// TIA Portal project "automated-warehouse" (V18)
// Vorlageprojekt für das Buch mit Zielsystem S7-1200

(* hardware
DEVICE "S7-1200-Station_1"  S7-1200 Station
   slot 0: "Baugruppenträger_0"  Rack  V1.0
   slot 1: "PLC_1"  CPU 1211C DC/DC/DC  6ES7 211-1AE40-0XB0  V4.1
*)

// ===== PLC "PLC_1"  CPU 1211C DC/DC/DC =====

VAR_GLOBAL   // PLC tag table "Standard-Variablentabelle"
   "Stored Shelf Value" AT %MW0 : Int;
   "Load Sequence Active" AT %M0.1 : Bool;
   "Unload Sequence Active" AT %M0.2 : Bool;
END_VAR

VAR_GLOBAL   // PLC tag table "FactoryIO"
   "Lift" AT %Q0.4 : Bool;
   "Forks Left" AT %Q0.2 : Bool;
   "Forks Right" AT %Q0.3 : Bool;
   "Entry Conveyor" AT %Q0.0 : Bool;
   "Load Conveyor" AT %Q0.1 : Bool;
   "Unload Conveyor" AT %Q0.5 : Bool;
   "Exit Conveyor" AT %Q0.6 : Bool;
   "Start light" AT %Q0.7 : Bool;
   "Stop light" AT %Q1.1 : Bool;
   "Target Position" AT %QD30 : DInt;
   "Reset Light" AT %Q1.0 : Bool;
   "At Entry" AT %I0.0 : Bool;
   "At Load" AT %I0.1 : Bool;
   "At Left" AT %I0.2 : Bool;
   "At Middle" AT %I0.3 : Bool;
   "At Right" AT %I0.4 : Bool;
   "At Unload" AT %I0.5 : Bool;
   "At Exit" AT %I0.6 : Bool;
   "Moving X" AT %I0.7 : Bool;
   "Moving Z" AT %I1.0 : Bool;
   "Start" AT %I1.1 : Bool;
   "Reset" AT %I1.2 : Bool;
   "Stop" AT %I1.3 : Bool;
   "Emergency stop" AT %I1.4 : Bool;
   "Load mode" AT %I1.5 : Bool;
END_VAR

DATA_BLOCK "Stacker Crane_DB"   // DB1
{ S7_Optimized_Access := 'TRUE' }
VERSION : 0.1
// stored: InstanceOfName Stacker Crane
"Stacker Crane"
BEGIN
END_DATA_BLOCK

DATA_BLOCK "Control Panel_DB"   // DB2
{ S7_Optimized_Access := 'TRUE' }
VERSION : 0.1
// stored: InstanceOfName Control Panel
"Control Panel"
BEGIN
END_DATA_BLOCK

DATA_BLOCK "Conveyors_DB"   // DB3
{ S7_Optimized_Access := 'TRUE' }
VERSION : 0.1
// stored: InstanceOfName Conveyors
"Conveyors"
BEGIN
END_DATA_BLOCK

// folder: System blocks/Program resources

DATA_BLOCK "IEC_Timer_0_DB"   // DB4
{ S7_Optimized_Access := 'TRUE' }
AUTHOR : Simatic
FAMILY : IEC
NAME : IEC_TMR
VERSION : 1.0
// stored: InstanceOfName IEC_TIMER
"IEC_TIMER"
BEGIN
END_DATA_BLOCK

DATA_BLOCK "IEC_Timer_0_DB_1"   // DB5
{ S7_Optimized_Access := 'TRUE' }
AUTHOR : Simatic
FAMILY : IEC
NAME : IEC_TMR
VERSION : 1.0
// stored: InstanceOfName IEC_TIMER
"IEC_TIMER"
BEGIN
END_DATA_BLOCK

// folder: (top level)

FUNCTION_BLOCK "Stacker Crane"   // FB1, LAD
{ S7_Optimized_Access := 'TRUE' }
VERSION : 0.1
   VAR_INPUT
      "Moving X" : Bool;
      "Moving Z" : Bool;
      "At Entry" : Bool;
      "At Load" : Bool;
      "At Unload" : Bool;
      "At Left" : Bool;
      "At Middle" : Bool;
      "At Right" : Bool;
      "Load mode" : Bool;
      Reset : Bool;
      "Start light" : Bool;
      "Emergency Stop" : Bool;
   END_VAR
   VAR_OUTPUT
      Lift : Bool;
      "Forks Left" : Bool;
      "Forks Right" : Bool;
      "Target Position" : DInt;
      "Stored Shelf Value" : Int;
      "Load Sequence Active" : Bool;
      "Unload Sequence Active" : Bool;
   END_VAR
   VAR
      n_trig : Array[0..10] of Bool;
      "Step" : Int := 0;
   END_VAR
   VAR_TEMP   // added for the SCL form of the ladder/FBD networks
      _w1 : Bool;
      _w2 : Bool;
      _w3 : Bool;
   END_VAR
BEGIN

REGION Network 1: <-------------------------- Load Section -------------------------->
END_REGION

REGION Network 2: Step 0 - Start Load Sequence
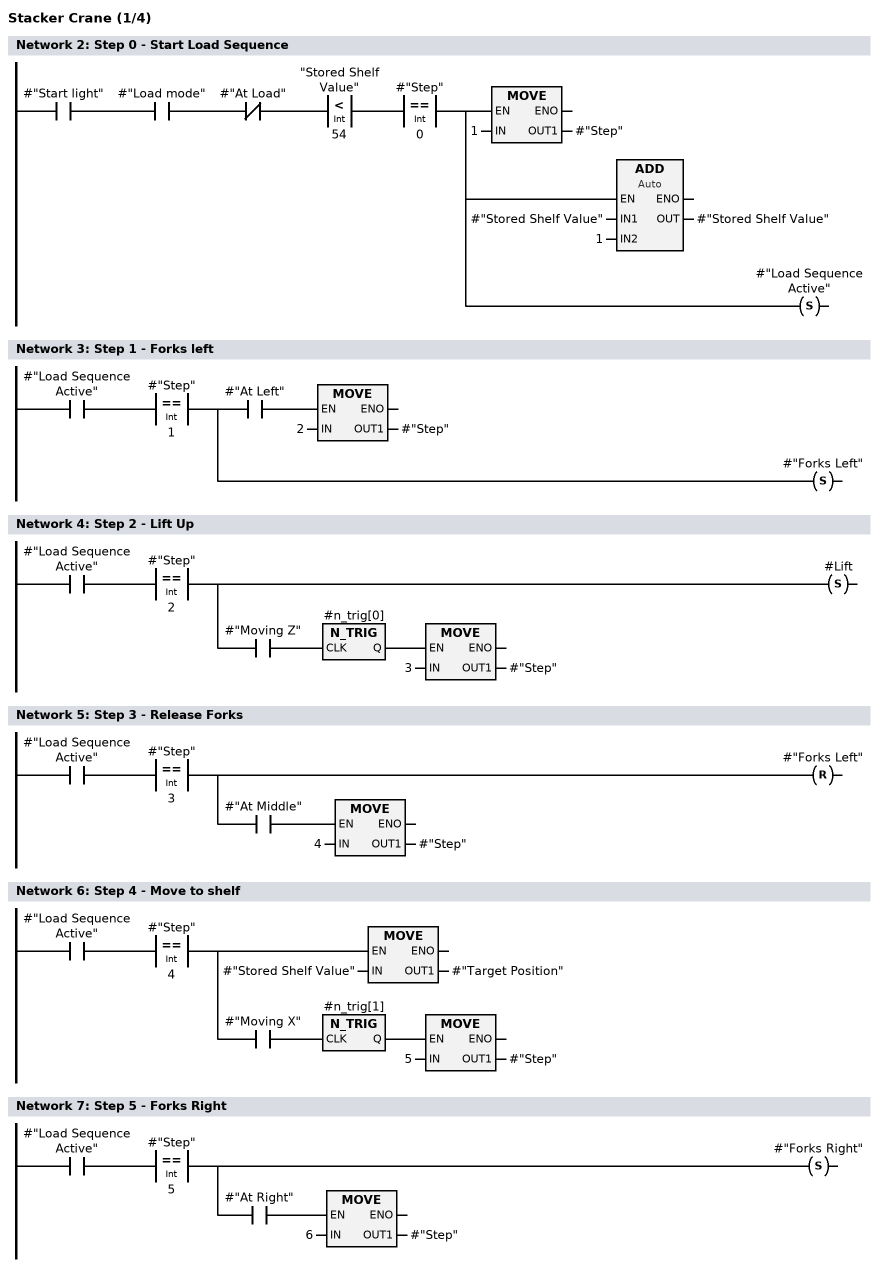
   RUNG wire#powerrail
      Contact( #"Start light" )
      Contact( #"Load mode" )
      I_Contact( #"At Load" )
      { S7_Templates := "SrcType := Int" } LT_Contact(in1 := "Stored Shelf Value", in2 := 54)
      { S7_Templates := "SrcType := Int" } EQ_Contact(in1 := #"Step", in2 := 0)
      wire#w1
      Move(in := 1, out1 => #"Step")
   END_RUNG
   RUNG wire#w1
      Add(in1 := #"Stored Shelf Value", in2 := 1, out => #"Stored Shelf Value")
   END_RUNG
   RUNG wire#w1
      S_Coil( #"Load Sequence Active" )
   END_RUNG
   // the same network as SCL:
   #_w1 := #"Start light" AND #"Load mode" AND NOT #"At Load" AND ("Stored Shelf Value" < 54) AND (#"Step" = 0);
   IF #_w1 THEN
       #"Step" := 1;
       #"Stored Shelf Value" := #"Stored Shelf Value" + 1;
       #"Load Sequence Active" := TRUE;
   END_IF;
END_REGION

REGION Network 3: Step 1 - Forks left
   RUNG wire#powerrail
      Contact( #"Load Sequence Active" )
      { S7_Templates := "SrcType := Int" } EQ_Contact(in1 := #"Step", in2 := 1)
      wire#w1
      Contact( #"At Left" )
      Move(in := 2, out1 => #"Step")
   END_RUNG
   RUNG wire#w1
      S_Coil( #"Forks Left" )
   END_RUNG
   // the same network as SCL:
   #_w1 := #"Load Sequence Active" AND (#"Step" = 1);
   IF #_w1 AND #"At Left" THEN #"Step" := 2; END_IF;
   IF #_w1 THEN #"Forks Left" := TRUE; END_IF;
END_REGION

REGION Network 4: Step 2 - Lift Up
   RUNG wire#powerrail
      Contact( #"Load Sequence Active" )
      { S7_Templates := "SrcType := Int" } EQ_Contact(in1 := #"Step", in2 := 2)
      wire#w1
      S_Coil( #Lift )
   END_RUNG
   RUNG wire#w1
      Contact( #"Moving Z" )
      N_Trig( #n_trig[0] )
      Move(in := 3, out1 => #"Step")
   END_RUNG
   // the same network as SCL:
   #_w1 := #"Load Sequence Active" AND (#"Step" = 2);
   IF #_w1 THEN #Lift := TRUE; END_IF;
   #_w2 := #_w1 AND #"Moving Z";
   #_w3 := NOT #_w2 AND #n_trig[0];   // falling edge
   #n_trig[0] := #_w2;
   IF #_w3 THEN #"Step" := 3; END_IF;
END_REGION

REGION Network 5: Step 3 - Release Forks
   RUNG wire#powerrail
      Contact( #"Load Sequence Active" )
      { S7_Templates := "SrcType := Int" } EQ_Contact(in1 := #"Step", in2 := 3)
      wire#w1
      R_Coil( #"Forks Left" )
   END_RUNG
   RUNG wire#w1
      Contact( #"At Middle" )
      Move(in := 4, out1 => #"Step")
   END_RUNG
   // the same network as SCL:
   #_w1 := #"Load Sequence Active" AND (#"Step" = 3);
   IF #_w1 THEN #"Forks Left" := FALSE; END_IF;
   IF #_w1 AND #"At Middle" THEN #"Step" := 4; END_IF;
END_REGION

REGION Network 6: Step 4 - Move to shelf
   RUNG wire#powerrail
      Contact( #"Load Sequence Active" )
      { S7_Templates := "SrcType := Int" } EQ_Contact(in1 := #"Step", in2 := 4)
      wire#w1
      Move(in := #"Stored Shelf Value", out1 => #"Target Position")
   END_RUNG
   RUNG wire#w1
      Contact( #"Moving X" )
      N_Trig( #n_trig[1] )
      Move(in := 5, out1 => #"Step")
   END_RUNG
   // the same network as SCL:
   #_w1 := #"Load Sequence Active" AND (#"Step" = 4);
   IF #_w1 THEN #"Target Position" := #"Stored Shelf Value"; END_IF;
   #_w2 := #_w1 AND #"Moving X";
   #_w3 := NOT #_w2 AND #n_trig[1];   // falling edge
   #n_trig[1] := #_w2;
   IF #_w3 THEN #"Step" := 5; END_IF;
END_REGION

REGION Network 7: Step 5 - Forks Right
   RUNG wire#powerrail
      Contact( #"Load Sequence Active" )
      { S7_Templates := "SrcType := Int" } EQ_Contact(in1 := #"Step", in2 := 5)
      wire#w1
      S_Coil( #"Forks Right" )
   END_RUNG
   RUNG wire#w1
      Contact( #"At Right" )
      Move(in := 6, out1 => #"Step")
   END_RUNG
   // the same network as SCL:
   #_w1 := #"Load Sequence Active" AND (#"Step" = 5);
   IF #_w1 THEN #"Forks Right" := TRUE; END_IF;
   IF #_w1 AND #"At Right" THEN #"Step" := 6; END_IF;
END_REGION

REGION Network 8: Step 6 - Release Lift
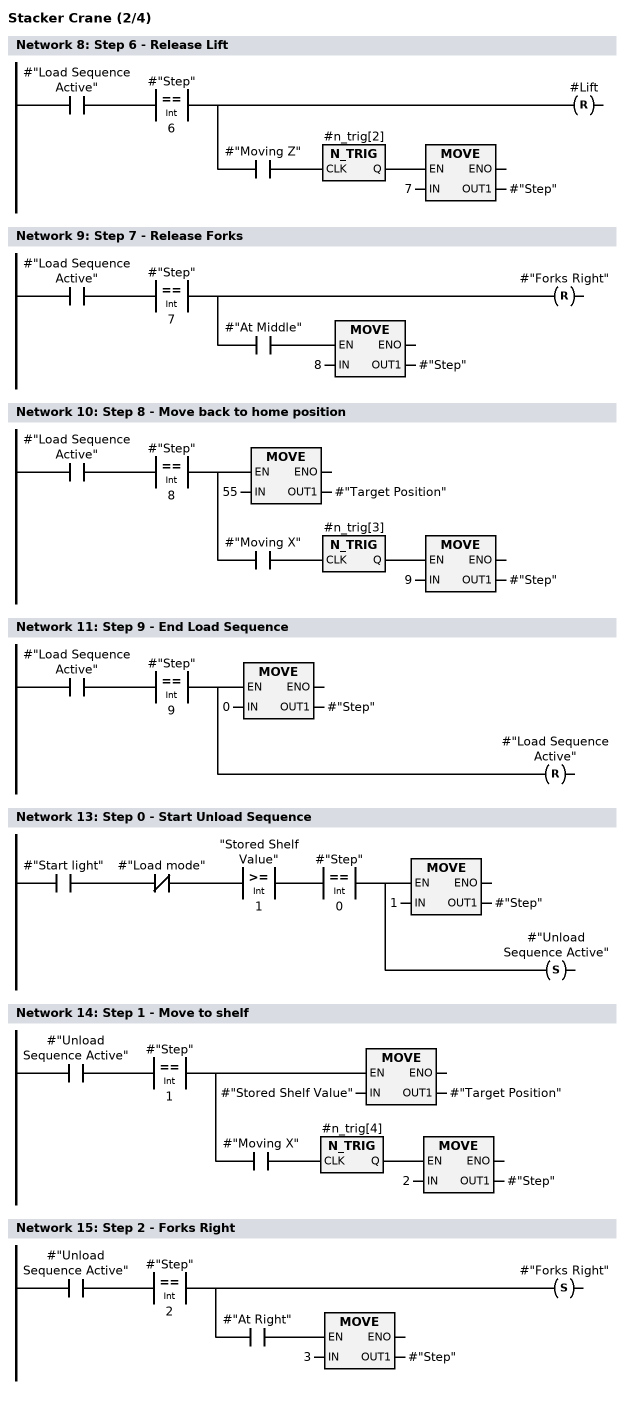
   RUNG wire#powerrail
      Contact( #"Load Sequence Active" )
      { S7_Templates := "SrcType := Int" } EQ_Contact(in1 := #"Step", in2 := 6)
      wire#w1
      R_Coil( #Lift )
   END_RUNG
   RUNG wire#w1
      Contact( #"Moving Z" )
      N_Trig( #n_trig[2] )
      Move(in := 7, out1 => #"Step")
   END_RUNG
   // the same network as SCL:
   #_w1 := #"Load Sequence Active" AND (#"Step" = 6);
   IF #_w1 THEN #Lift := FALSE; END_IF;
   #_w2 := #_w1 AND #"Moving Z";
   #_w3 := NOT #_w2 AND #n_trig[2];   // falling edge
   #n_trig[2] := #_w2;
   IF #_w3 THEN #"Step" := 7; END_IF;
END_REGION

REGION Network 9: Step 7 - Release Forks
   RUNG wire#powerrail
      Contact( #"Load Sequence Active" )
      { S7_Templates := "SrcType := Int" } EQ_Contact(in1 := #"Step", in2 := 7)
      wire#w1
      R_Coil( #"Forks Right" )
   END_RUNG
   RUNG wire#w1
      Contact( #"At Middle" )
      Move(in := 8, out1 => #"Step")
   END_RUNG
   // the same network as SCL:
   #_w1 := #"Load Sequence Active" AND (#"Step" = 7);
   IF #_w1 THEN #"Forks Right" := FALSE; END_IF;
   IF #_w1 AND #"At Middle" THEN #"Step" := 8; END_IF;
END_REGION

REGION Network 10: Step 8 - Move back to home position
   RUNG wire#powerrail
      Contact( #"Load Sequence Active" )
      { S7_Templates := "SrcType := Int" } EQ_Contact(in1 := #"Step", in2 := 8)
      wire#w1
      Move(in := 55, out1 => #"Target Position")
   END_RUNG
   RUNG wire#w1
      Contact( #"Moving X" )
      N_Trig( #n_trig[3] )
      Move(in := 9, out1 => #"Step")
   END_RUNG
   // the same network as SCL:
   #_w1 := #"Load Sequence Active" AND (#"Step" = 8);
   IF #_w1 THEN #"Target Position" := 55; END_IF;
   #_w2 := #_w1 AND #"Moving X";
   #_w3 := NOT #_w2 AND #n_trig[3];   // falling edge
   #n_trig[3] := #_w2;
   IF #_w3 THEN #"Step" := 9; END_IF;
END_REGION

REGION Network 11: Step 9 - End Load Sequence
   RUNG wire#powerrail
      Contact( #"Load Sequence Active" )
      { S7_Templates := "SrcType := Int" } EQ_Contact(in1 := #"Step", in2 := 9)
      wire#w1
      Move(in := 0, out1 => #"Step")
   END_RUNG
   RUNG wire#w1
      R_Coil( #"Load Sequence Active" )
   END_RUNG
   // the same network as SCL:
   #_w1 := #"Load Sequence Active" AND (#"Step" = 9);
   IF #_w1 THEN
       #"Step" := 0;
       #"Load Sequence Active" := FALSE;
   END_IF;
END_REGION

REGION Network 12: <-------------------------- Unload Section -------------------------->
END_REGION

REGION Network 13: Step 0 - Start Unload Sequence
   RUNG wire#powerrail
      Contact( #"Start light" )
      I_Contact( #"Load mode" )
      { S7_Templates := "SrcType := Int" } GE_Contact(in1 := "Stored Shelf Value", in2 := 1)
      { S7_Templates := "SrcType := Int" } EQ_Contact(in1 := #"Step", in2 := 0)
      wire#w1
      Move(in := 1, out1 => #"Step")
   END_RUNG
   RUNG wire#w1
      S_Coil( #"Unload Sequence Active" )
   END_RUNG
   // the same network as SCL:
   #_w1 := #"Start light" AND NOT #"Load mode" AND ("Stored Shelf Value" >= 1) AND (#"Step" = 0);
   IF #_w1 THEN
       #"Step" := 1;
       #"Unload Sequence Active" := TRUE;
   END_IF;
END_REGION

REGION Network 14: Step 1 - Move to shelf
   RUNG wire#powerrail
      Contact( #"Unload Sequence Active" )
      { S7_Templates := "SrcType := Int" } EQ_Contact(in1 := #"Step", in2 := 1)
      wire#w1
      Move(in := #"Stored Shelf Value", out1 => #"Target Position")
   END_RUNG
   RUNG wire#w1
      Contact( #"Moving X" )
      N_Trig( #n_trig[4] )
      Move(in := 2, out1 => #"Step")
   END_RUNG
   // the same network as SCL:
   #_w1 := #"Unload Sequence Active" AND (#"Step" = 1);
   IF #_w1 THEN #"Target Position" := #"Stored Shelf Value"; END_IF;
   #_w2 := #_w1 AND #"Moving X";
   #_w3 := NOT #_w2 AND #n_trig[4];   // falling edge
   #n_trig[4] := #_w2;
   IF #_w3 THEN #"Step" := 2; END_IF;
END_REGION

REGION Network 15: Step 2 - Forks Right
   RUNG wire#powerrail
      Contact( #"Unload Sequence Active" )
      { S7_Templates := "SrcType := Int" } EQ_Contact(in1 := #"Step", in2 := 2)
      wire#w1
      S_Coil( #"Forks Right" )
   END_RUNG
   RUNG wire#w1
      Contact( #"At Right" )
      Move(in := 3, out1 => #"Step")
   END_RUNG
   // the same network as SCL:
   #_w1 := #"Unload Sequence Active" AND (#"Step" = 2);
   IF #_w1 THEN #"Forks Right" := TRUE; END_IF;
   IF #_w1 AND #"At Right" THEN #"Step" := 3; END_IF;
END_REGION

REGION Network 16: Step 3 - Lift Up
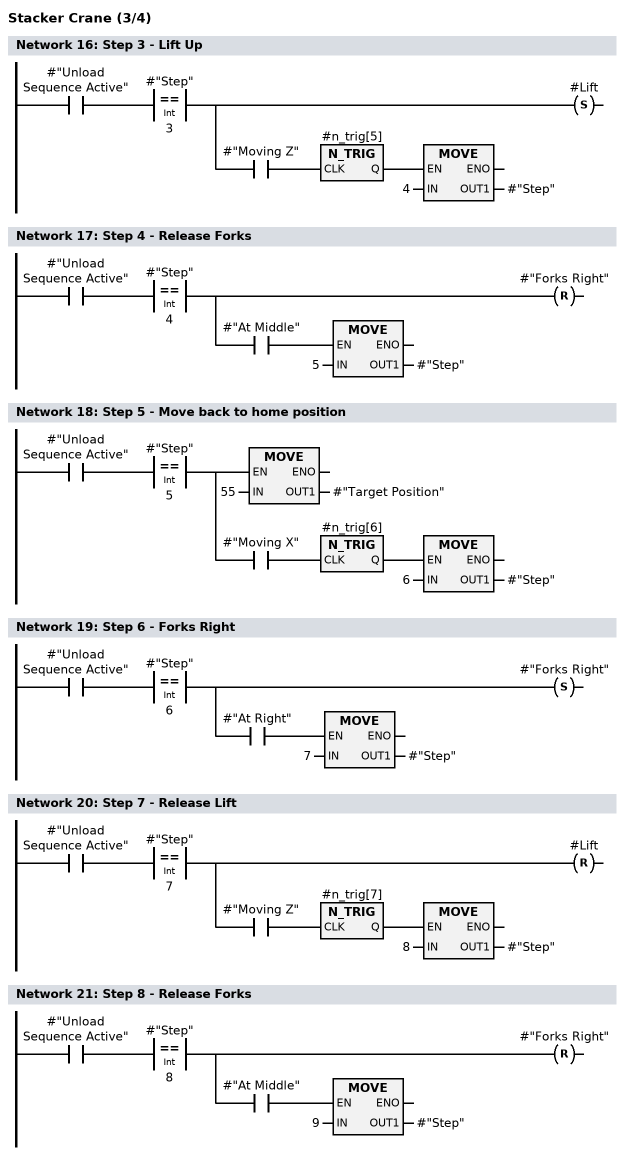
   RUNG wire#powerrail
      Contact( #"Unload Sequence Active" )
      { S7_Templates := "SrcType := Int" } EQ_Contact(in1 := #"Step", in2 := 3)
      wire#w1
      S_Coil( #Lift )
   END_RUNG
   RUNG wire#w1
      Contact( #"Moving Z" )
      N_Trig( #n_trig[5] )
      Move(in := 4, out1 => #"Step")
   END_RUNG
   // the same network as SCL:
   #_w1 := #"Unload Sequence Active" AND (#"Step" = 3);
   IF #_w1 THEN #Lift := TRUE; END_IF;
   #_w2 := #_w1 AND #"Moving Z";
   #_w3 := NOT #_w2 AND #n_trig[5];   // falling edge
   #n_trig[5] := #_w2;
   IF #_w3 THEN #"Step" := 4; END_IF;
END_REGION

REGION Network 17: Step 4 - Release Forks
   RUNG wire#powerrail
      Contact( #"Unload Sequence Active" )
      { S7_Templates := "SrcType := Int" } EQ_Contact(in1 := #"Step", in2 := 4)
      wire#w1
      R_Coil( #"Forks Right" )
   END_RUNG
   RUNG wire#w1
      Contact( #"At Middle" )
      Move(in := 5, out1 => #"Step")
   END_RUNG
   // the same network as SCL:
   #_w1 := #"Unload Sequence Active" AND (#"Step" = 4);
   IF #_w1 THEN #"Forks Right" := FALSE; END_IF;
   IF #_w1 AND #"At Middle" THEN #"Step" := 5; END_IF;
END_REGION

REGION Network 18: Step 5 - Move back to home position
   RUNG wire#powerrail
      Contact( #"Unload Sequence Active" )
      { S7_Templates := "SrcType := Int" } EQ_Contact(in1 := #"Step", in2 := 5)
      wire#w1
      Move(in := 55, out1 => #"Target Position")
   END_RUNG
   RUNG wire#w1
      Contact( #"Moving X" )
      N_Trig( #n_trig[6] )
      Move(in := 6, out1 => #"Step")
   END_RUNG
   // the same network as SCL:
   #_w1 := #"Unload Sequence Active" AND (#"Step" = 5);
   IF #_w1 THEN #"Target Position" := 55; END_IF;
   #_w2 := #_w1 AND #"Moving X";
   #_w3 := NOT #_w2 AND #n_trig[6];   // falling edge
   #n_trig[6] := #_w2;
   IF #_w3 THEN #"Step" := 6; END_IF;
END_REGION

REGION Network 19: Step 6 - Forks Right
   RUNG wire#powerrail
      Contact( #"Unload Sequence Active" )
      { S7_Templates := "SrcType := Int" } EQ_Contact(in1 := #"Step", in2 := 6)
      wire#w1
      S_Coil( #"Forks Right" )
   END_RUNG
   RUNG wire#w1
      Contact( #"At Right" )
      Move(in := 7, out1 => #"Step")
   END_RUNG
   // the same network as SCL:
   #_w1 := #"Unload Sequence Active" AND (#"Step" = 6);
   IF #_w1 THEN #"Forks Right" := TRUE; END_IF;
   IF #_w1 AND #"At Right" THEN #"Step" := 7; END_IF;
END_REGION

REGION Network 20: Step 7 - Release Lift
   RUNG wire#powerrail
      Contact( #"Unload Sequence Active" )
      { S7_Templates := "SrcType := Int" } EQ_Contact(in1 := #"Step", in2 := 7)
      wire#w1
      R_Coil( #Lift )
   END_RUNG
   RUNG wire#w1
      Contact( #"Moving Z" )
      N_Trig( #n_trig[7] )
      Move(in := 8, out1 => #"Step")
   END_RUNG
   // the same network as SCL:
   #_w1 := #"Unload Sequence Active" AND (#"Step" = 7);
   IF #_w1 THEN #Lift := FALSE; END_IF;
   #_w2 := #_w1 AND #"Moving Z";
   #_w3 := NOT #_w2 AND #n_trig[7];   // falling edge
   #n_trig[7] := #_w2;
   IF #_w3 THEN #"Step" := 8; END_IF;
END_REGION

REGION Network 21: Step 8 - Release Forks
   RUNG wire#powerrail
      Contact( #"Unload Sequence Active" )
      { S7_Templates := "SrcType := Int" } EQ_Contact(in1 := #"Step", in2 := 8)
      wire#w1
      R_Coil( #"Forks Right" )
   END_RUNG
   RUNG wire#w1
      Contact( #"At Middle" )
      Move(in := 9, out1 => #"Step")
   END_RUNG
   // the same network as SCL:
   #_w1 := #"Unload Sequence Active" AND (#"Step" = 8);
   IF #_w1 THEN #"Forks Right" := FALSE; END_IF;
   IF #_w1 AND #"At Middle" THEN #"Step" := 9; END_IF;
END_REGION

REGION Network 22: Step 9 - End Load Sequence
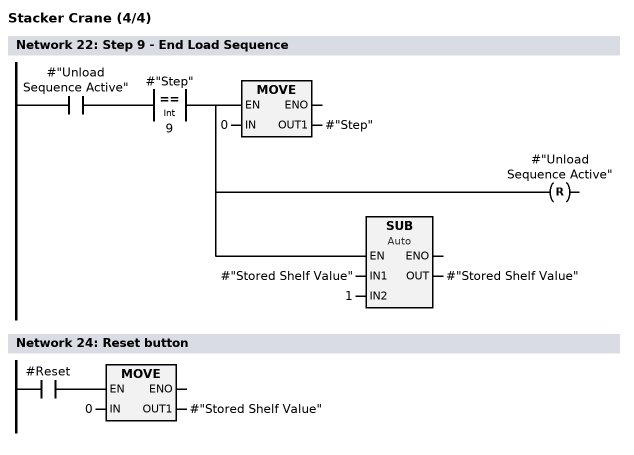
   RUNG wire#powerrail
      Contact( #"Unload Sequence Active" )
      { S7_Templates := "SrcType := Int" } EQ_Contact(in1 := #"Step", in2 := 9)
      wire#w1
      Move(in := 0, out1 => #"Step")
   END_RUNG
   RUNG wire#w1
      R_Coil( #"Unload Sequence Active" )
   END_RUNG
   RUNG wire#w1
      Sub(in1 := #"Stored Shelf Value", in2 := 1, out => #"Stored Shelf Value")
   END_RUNG
   // the same network as SCL:
   #_w1 := #"Unload Sequence Active" AND (#"Step" = 9);
   IF #_w1 THEN
       #"Step" := 0;
       #"Unload Sequence Active" := FALSE;
       #"Stored Shelf Value" := #"Stored Shelf Value" - 1;
   END_IF;
END_REGION

REGION Network 23: <-------------------------- Buttons Section -------------------------->
END_REGION

REGION Network 24: Reset button
   RUNG wire#powerrail
      Contact( #Reset )
      Move(in := 0, out1 => #"Stored Shelf Value")
   END_RUNG
   // the same network as SCL:
   IF #Reset THEN #"Stored Shelf Value" := 0; END_IF;
END_REGION

REGION Network 25: Emergency stop
END_REGION
END_FUNCTION_BLOCK

FUNCTION_BLOCK "Conveyors"   // FB2, LAD
{ S7_Optimized_Access := 'TRUE' }
VERSION : 0.1
   VAR_INPUT
      "At Entry" : Bool;
      "At Load" : Bool;
      "At Unload" : Bool;
      "Stored Shelf Value" : Int;
      "At Exit" : Bool;
   END_VAR
   VAR_OUTPUT
      "Entry Conveyor" : Bool;
      "Load Conveyor" : Bool;
      "Unload Conveyor" : Bool;
      "Exit Conveyor" : Bool;
   END_VAR
BEGIN

REGION Network 1: Entry Conveyor
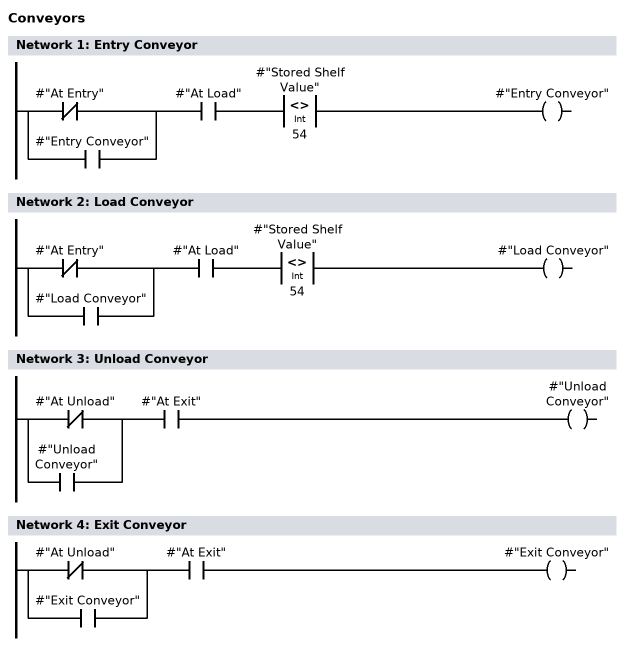
   RUNG wire#powerrail
      I_Contact( #"At Entry" )
      wire#w1
      Contact( #"At Load" )
      { S7_Templates := "SrcType := Int" } NE_Contact(in1 := #"Stored Shelf Value", in2 := 54)
      Coil( #"Entry Conveyor" )
   END_RUNG
   RUNG wire#powerrail
      Contact( #"Entry Conveyor" )
   END_RUNG wire#w1
   // the same network as SCL:
   #"Entry Conveyor" := (NOT #"At Entry" OR #"Entry Conveyor") AND #"At Load" AND (#"Stored Shelf Value" <> 54);
END_REGION

REGION Network 2: Load Conveyor
   RUNG wire#powerrail
      I_Contact( #"At Entry" )
      wire#w1
      Contact( #"At Load" )
      { S7_Templates := "SrcType := Int" } NE_Contact(in1 := #"Stored Shelf Value", in2 := 54)
      Coil( #"Load Conveyor" )
   END_RUNG
   RUNG wire#powerrail
      Contact( #"Load Conveyor" )
   END_RUNG wire#w1
   // the same network as SCL:
   #"Load Conveyor" := (NOT #"At Entry" OR #"Load Conveyor") AND #"At Load" AND (#"Stored Shelf Value" <> 54);
END_REGION

REGION Network 3: Unload Conveyor
   RUNG wire#powerrail
      I_Contact( #"At Unload" )
      wire#w1
      Contact( #"At Exit" )
      Coil( #"Unload Conveyor" )
   END_RUNG
   RUNG wire#powerrail
      Contact( #"Unload Conveyor" )
   END_RUNG wire#w1
   // the same network as SCL:
   #"Unload Conveyor" := (NOT #"At Unload" OR #"Unload Conveyor") AND #"At Exit";
END_REGION

REGION Network 4: Exit Conveyor
   RUNG wire#powerrail
      I_Contact( #"At Unload" )
      wire#w1
      Contact( #"At Exit" )
      Coil( #"Exit Conveyor" )
   END_RUNG
   RUNG wire#powerrail
      Contact( #"Exit Conveyor" )
   END_RUNG wire#w1
   // the same network as SCL:
   #"Exit Conveyor" := (NOT #"At Unload" OR #"Exit Conveyor") AND #"At Exit";
END_REGION
END_FUNCTION_BLOCK

FUNCTION_BLOCK "Control Panel"   // FB3, LAD
{ S7_Optimized_Access := 'TRUE' }
VERSION : 0.1
   VAR_INPUT
      Start : Bool;
      Reset : Bool;
      Stop : Bool;
      "Emergency stop" : Bool;
      "Unload Sequence Active" : Bool;
      "Load Sequence Active" : Bool;
      "Stored Shelf Value" : Int;
   END_VAR
   VAR_OUTPUT
      "Start light" : Bool;
      "Reset light" : Bool;
      "Stop light" : Bool;
   END_VAR
   VAR
      n_trig : Array[0..3] of Bool;
   END_VAR
   VAR_TEMP   // added for the SCL form of the ladder/FBD networks
      _w1 : Bool;
      _w2 : Bool;
   END_VAR
BEGIN

REGION Network 1: Start
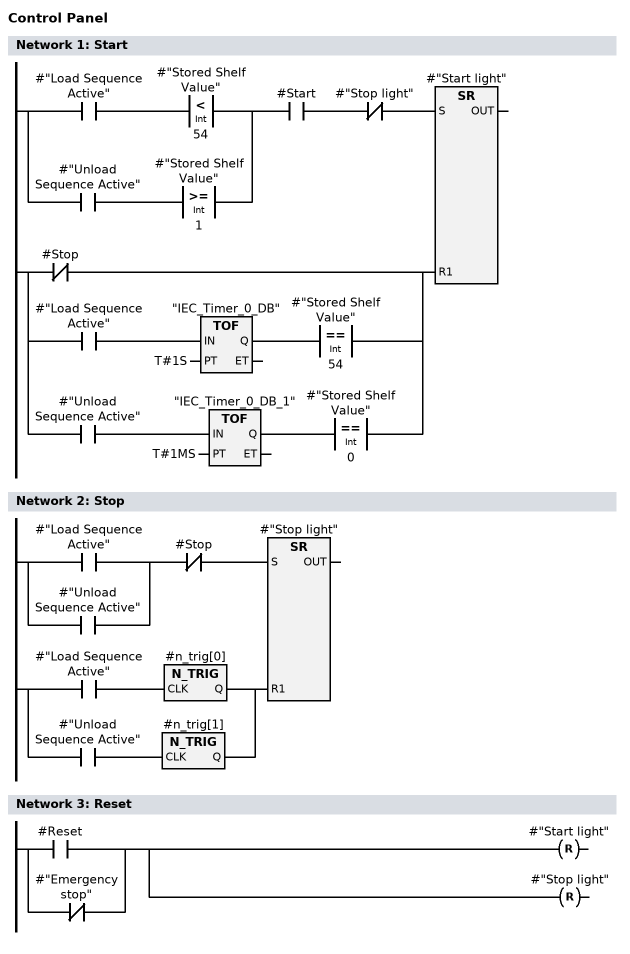
   "IEC_Timer_0_DB".TOF(IN := #"Load Sequence Active", PT := T#1S);
   "IEC_Timer_0_DB_1".TOF(IN := #"Unload Sequence Active", PT := T#1MS);
   IF ((#"Load Sequence Active" AND (#"Stored Shelf Value" < 54)) OR (#"Unload Sequence Active" AND (#"Stored Shelf Value" >= 1))) AND #Start AND NOT #"Stop light" THEN
       #"Start light" := TRUE;   // SR flip-flop
   END_IF;
   IF NOT #Stop OR ("IEC_Timer_0_DB".Q AND (#"Stored Shelf Value" = 54)) OR ("IEC_Timer_0_DB_1".Q AND (#"Stored Shelf Value" = 0)) THEN
       #"Start light" := FALSE;
   END_IF;
END_REGION

REGION Network 2: Stop
   RUNG wire#powerrail
      Contact( #"Load Sequence Active" )
      wire#w1
      I_Contact( #Stop )
      S_SR(operand := #"Stop light", r1 := wire#w2)
   END_RUNG
   RUNG wire#powerrail
      Contact( #"Unload Sequence Active" )
   END_RUNG wire#w1
   RUNG wire#powerrail
      Contact( #"Load Sequence Active" )
      N_Trig( #n_trig[0] )
   END_RUNG wire#w2
   RUNG wire#powerrail
      Contact( #"Unload Sequence Active" )
      N_Trig( #n_trig[1] )
   END_RUNG wire#w2
   // the same network as SCL:
   #_w1 := NOT #"Load Sequence Active" AND #n_trig[0];   // falling edge
   #n_trig[0] := #"Load Sequence Active";
   #_w2 := NOT #"Unload Sequence Active" AND #n_trig[1];   // falling edge
   #n_trig[1] := #"Unload Sequence Active";
   IF (#"Load Sequence Active" OR #"Unload Sequence Active") AND NOT #Stop THEN
       #"Stop light" := TRUE;   // SR flip-flop
   END_IF;
   IF #_w1 OR #_w2 THEN #"Stop light" := FALSE; END_IF;
END_REGION

REGION Network 3: Reset
   RUNG wire#powerrail
      Contact( #Reset )
      wire#w1
      R_Coil( #"Start light" )
   END_RUNG
   RUNG wire#powerrail
      I_Contact( #"Emergency stop" )
   END_RUNG wire#w1
   RUNG wire#w1
      R_Coil( #"Stop light" )
   END_RUNG
   // the same network as SCL:
   IF #Reset OR NOT #"Emergency stop" THEN
       #"Start light" := FALSE;
       #"Stop light" := FALSE;
   END_IF;
END_REGION
END_FUNCTION_BLOCK

FUNCTION "MHJ-PLC-Lab-Function-S71200" : Void   // FC9000, SCL
{ S7_Optimized_Access := 'TRUE' }
VERSION : 0.1
   VAR_TEMP
      rdTimeReturn : Int;
      outputTime : DTL;
      SyncVal : Byte;
      forVal : Int;
      forVal_2 : Int;
      Value : Byte;
   END_VAR
   VAR CONSTANT
      CompVal : Byte := 16#34;
      Value_01 : Byte := 16#11;
      Value_01_DW : DWord := 16#A165_D992;
      Value_02_DW : DWord := 16#58BE_4401;
   END_VAR
BEGIN

   #Value:=PEEK(area := 16#82,
        dbNumber := 0,
        byteOffset := 511);
   #Value := #Value + 1;

   POKE(area := 16#82,
        dbNumber := 0,
        byteOffset := 511,
        value := #Value);

   POKE(area:=16#81,
        dbNumber:=0,
        byteOffset:=1016,
        value:=#Value_01_DW);
   POKE(area := 16#81,
        dbNumber := 0,
        byteOffset := 1020,
        value := #Value_02_DW);

   POKE(area := 16#81,
        dbNumber := 0,
        byteOffset := 511,
        value := B#16#00);

   FOR #forVal := 0 TO 120 DO
       FOR #forVal_2:=0 TO 10 DO
           #rdTimeReturn:=RD_SYS_T(#outputTime);
           #rdTimeReturn := WR_SYS_T(#outputTime);
           #rdTimeReturn := RD_SYS_T(#outputTime);
           #rdTimeReturn := WR_SYS_T(#outputTime);
       END_FOR;
       #SyncVal:= PEEK(area := 16#81,
                      dbNumber := 0,
                      byteOffset := 511);
       IF #SyncVal = #CompVal THEN
          GOTO M_1;
       END_IF;
   END_FOR;
   RETURN;

   M_1:
   POKE(area := 16#81,
        dbNumber := 0,
        byteOffset := 511,
        value := B#16#0);
END_FUNCTION

ORGANIZATION_BLOCK "Main"   // OB1, FBD, ProgramCycle
TITLE = "Main Program Sweep (Cycle)"
{ S7_Optimized_Access := 'TRUE' }
VERSION : 0.1
   VAR_INPUT
      Initial_Call : Bool;   // Initial call of this OB
      Remanence : Bool;   // =True, if remanent data are available
   END_VAR
BEGIN

REGION Network 1: Konnektierungsbaustein für PLC-Lab
   // Im Netzwerk 1 wird der Konnektierungsbaustein für PLC-Lab aufgerufen.
   // Dieser Aufruf darf nicht entfernt werden!
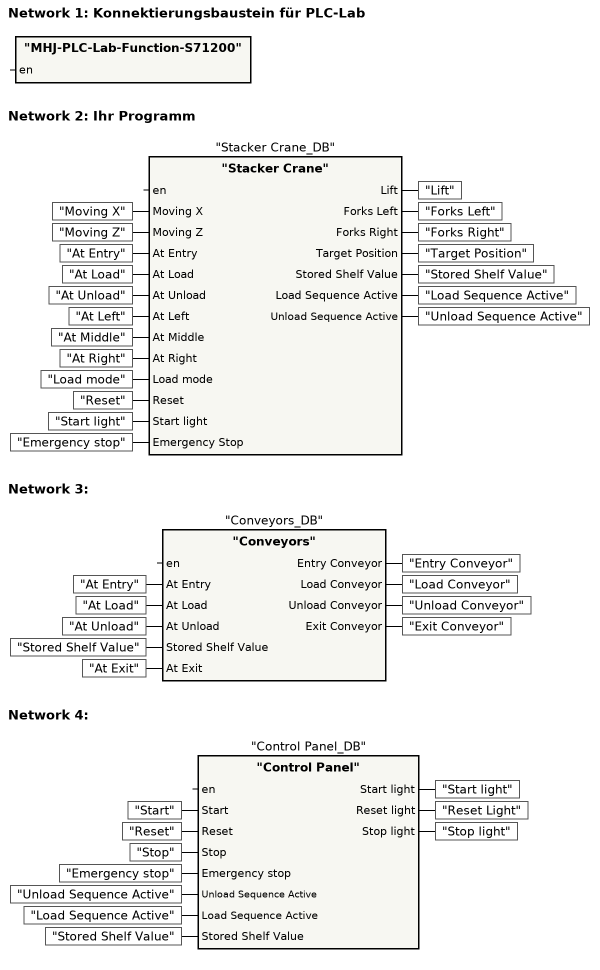
   "MHJ-PLC-Lab-Function-S71200"();
END_REGION

REGION Network 2: Ihr Programm
   // Schreiben Sie ab Netzwerk 2 Ihr Programm
   "Stacker Crane_DB"("Moving X" := "Moving X",   // "Stacker Crane"
                      "Moving Z" := "Moving Z",
                      "At Entry" := "At Entry",
                      "At Load" := "At Load",
                      "At Unload" := "At Unload",
                      "At Left" := "At Left",
                      "At Middle" := "At Middle",
                      "At Right" := "At Right",
                      "Load mode" := "Load mode",
                      Reset := "Reset",
                      "Start light" := "Start light",
                      "Emergency Stop" := "Emergency stop",
                      Lift => "Lift",
                      "Forks Left" => "Forks Left",
                      "Forks Right" => "Forks Right",
                      "Target Position" => "Target Position",
                      "Stored Shelf Value" => "Stored Shelf Value",
                      "Load Sequence Active" => "Load Sequence Active",
                      "Unload Sequence Active" => "Unload Sequence Active");
END_REGION

REGION Network 3
   "Conveyors_DB"("At Entry" := "At Entry",   // "Conveyors"
                  "At Load" := "At Load",
                  "At Unload" := "At Unload",
                  "Stored Shelf Value" := "Stored Shelf Value",
                  "At Exit" := "At Exit",
                  "Entry Conveyor" => "Entry Conveyor",
                  "Load Conveyor" => "Load Conveyor",
                  "Unload Conveyor" => "Unload Conveyor",
                  "Exit Conveyor" => "Exit Conveyor");
END_REGION

REGION Network 4
   "Control Panel_DB"(Start := "Start",   // "Control Panel"
                      Reset := "Reset",
                      Stop := "Stop",
                      "Emergency stop" := "Emergency stop",
                      "Unload Sequence Active" := "Unload Sequence Active",
                      "Load Sequence Active" := "Load Sequence Active",
                      "Stored Shelf Value" := "Stored Shelf Value",
                      "Start light" => "Start light",
                      "Reset light" => "Reset Light",
                      "Stop light" => "Stop light");
END_REGION
END_ORGANIZATION_BLOCK